// SIMATIC S7-200 SMART project (STEP 7-Micro/WIN SMART), CPU ST20

SYMBOL_TABLE USER1
IMaual           M1.0
IAuto            M1.1
QError           M1.2
UISetEnable1     M13.0
UIBtnExecute     M13.1
ConfigEpos1      VD608
UISetServeMode1  VW500
UISetServePos1   VD502
UISetMDI1        VD506
Positive1        V600.0
Negative1        V600.1
UISetJodForward1 V600.2
UISetJodReserve1 V600.3
UIBtnFlyRef1     V600.4   // 其他模式下回零
UISetResetErr1   V600.5
UISetOverV1      VW602    // 速度倍率（控制旋转快慢）
UISetOverAcc1    VW604    // 加速倍率（控制启动快慢）
UISetOverDec1    VW606    // 减速度倍率（控制停止快慢）
Axisenabled1     V650.0
AxisPosOk1       V650.1
AxisRef1         V650.2
Lockout1         V650.3
AxisWarn1        V650.4
AxisError1       V650.5
Overrange_Error1 V650.6
END_SYMBOL_TABLE

SYMBOL_TABLE 系统符号
Always_On        SM0.0    // 始终接通
First_Scan_On    SM0.1    // 仅在第一个扫描周期时接通
END_SYMBOL_TABLE

ORGANIZATION_BLOCK MAIN:OB1
TITLE=子程序注释
BEGIN
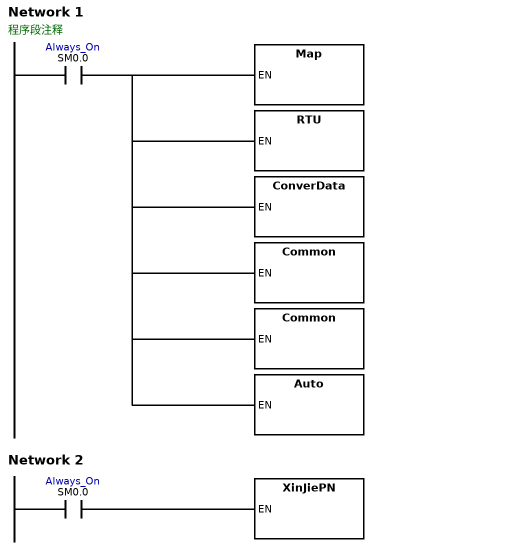
Network 1
// 程序段注释
LD     Always_On:SM0.0
CALL   Map:SBR5
CALL   RTU:SBR4
CALL   ConverData:SBR6
CALL   Common:SBR0
CALL   Common:SBR0
CALL   Auto:SBR3
Network 2
LD     Always_On:SM0.0
CALL   XinJiePN:SBR9
END_ORGANIZATION_BLOCK

// SBR1: protected block, not included

// SBR2: protected block, not included

SUBROUTINE_BLOCK RTU:SBR4
TITLE=子程序注释
VAR
tmpDone:BOOL;	// L0.0 
tmpErr:BYTE;	// LB1 
END_VAR
BEGIN
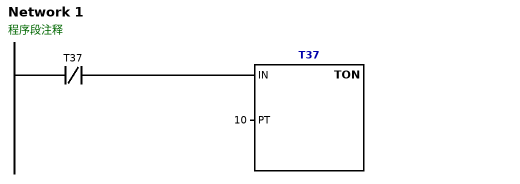
Network 1
// 程序段注释
LDN    T37
TON    T37, 10
END_SUBROUTINE_BLOCK

// SBR7: protected block, not included

// SBR8: protected block, not included

SUBROUTINE_BLOCK XinJiePN:SBR9
TITLE=子程序注释
VAR
tmpSpeed:DWORD;	// LD0 
tmpPos:DWORD;	// LD4 
tmpWarning:WORD;	// LW8 
tmpErr:WORD;	// LW10 
tmpDone:BOOL;	// L12.0 
tmpNotJOD:BOOL;	// L12.1 
END_VAR
BEGIN
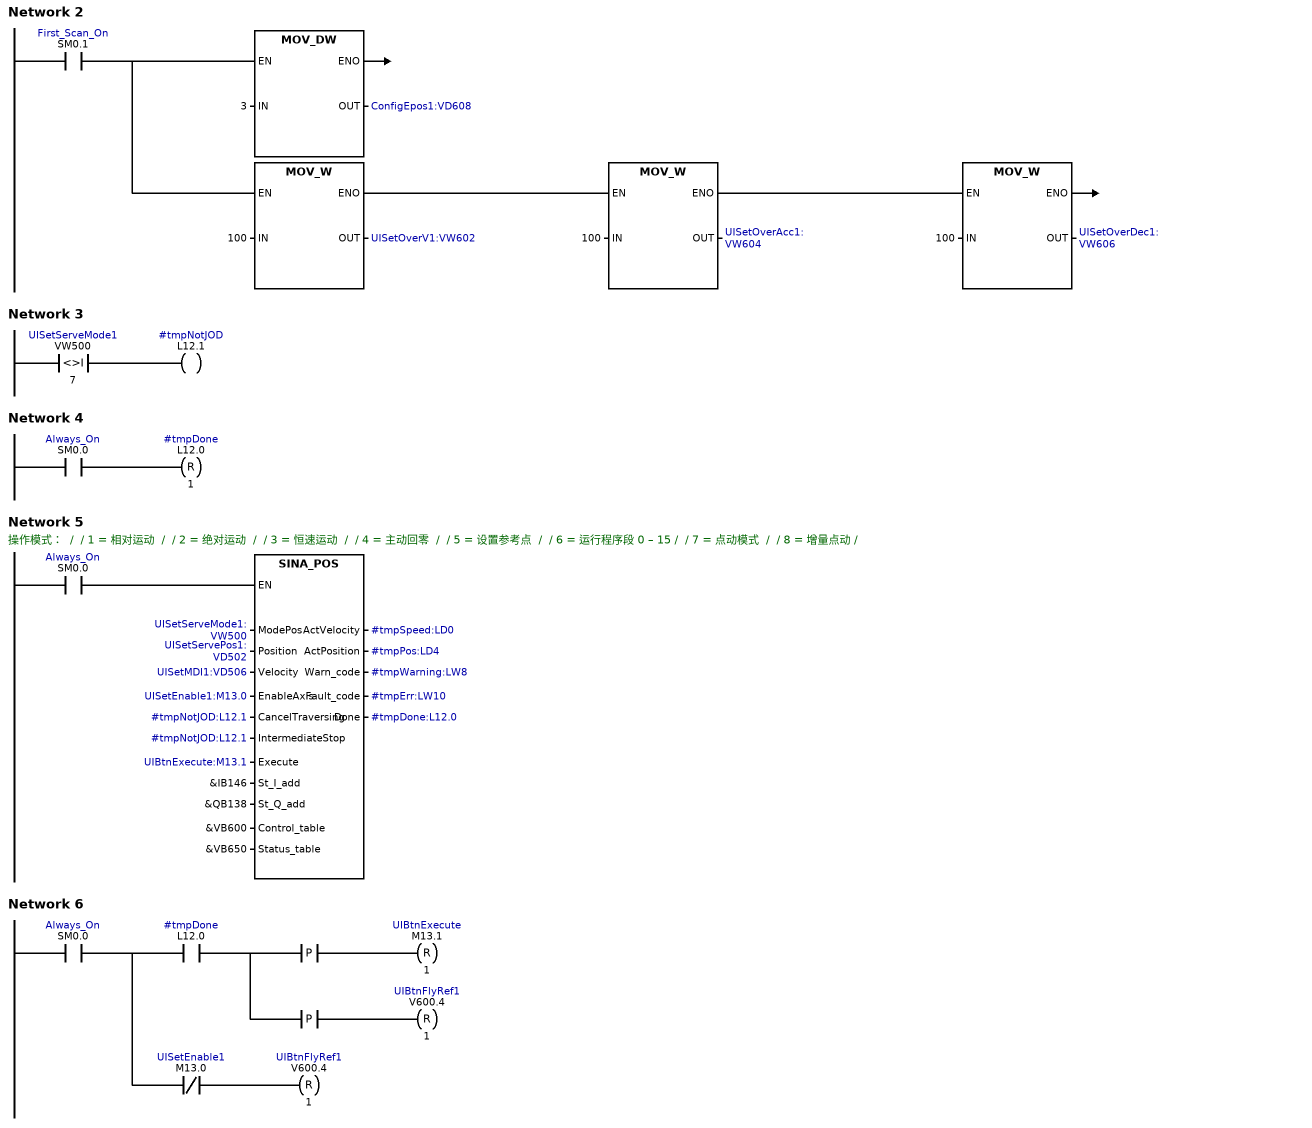
Network 2
LD     First_Scan_On:SM0.1
MOVD   3, ConfigEpos1:VD608
MOVW   100, UISetOverV1:VW602
AENO
MOVW   100, UISetOverAcc1:VW604
AENO
MOVW   100, UISetOverDec1:VW606
Network 3
LDW<>  UISetServeMode1:VW500, 7
=      #tmpNotJOD:L12.1
Network 4
LD     Always_On:SM0.0
R      #tmpDone:L12.0, 1
Network 5
// 操作模式： 
// 
// 1 = 相对运动 
// 
// 2 = 绝对运动 
// 
// 3 = 恒速运动 
// 
// 4 = 主动回零 
// 
// 5 = 设置参考点 
// 
// 6 = 运行程序段 0 – 15
// 
// 7 = 点动模式 
// 
// 8 = 增量点动
// 
LD     Always_On:SM0.0
CALL   SINA_POS:SBR8, UISetServeMode1:VW500, UISetServePos1:VD502, UISetMDI1:VD506, UISetEnable1:M13.0, #tmpNotJOD:L12.1, #tmpNotJOD:L12.1, UIBtnExecute:M13.1, &IB146, &QB138, &VB600, &VB650, #tmpSpeed:LD0, #tmpPos:LD4, #tmpWarning:LW8, #tmpErr:LW10, #tmpDone:L12.0
Network 6
LD     Always_On:SM0.0
LPS
A      #tmpDone:L12.0
LPS
EU
R      UIBtnExecute:M13.1, 1
LPP
EU
R      UIBtnFlyRef1:V600.4, 1
LPP
AN     UISetEnable1:M13.0
R      UIBtnFlyRef1:V600.4, 1
END_SUBROUTINE_BLOCK
